{attribute 'qualified_only'}
VAR_GLOBAL
	fJoystickLeftNormalizedY 		: LREAL;
	fJoystickLeftNormalizedX 		: LREAL;
	
	fJoystickRightNormalizedY 		: LREAL;
	fJoystickRightNormalizedX 		: LREAL;
	
	
	//fPositionCylPiston  		: LREAL;
	MCDirectionAxis1 : MC_Direction;
	MCDirectionAxis2 : MC_Direction;
	MCDirectionAxis3 : MC_Direction;
	MCDirectionAxis4 : MC_Direction;
	
		
END_VAR

(* stored: Version 1.1.0.1, ProductVersion 3.1.4024.12
   GVL G_Sensors: Id {d28c946e-63b0-41ab-8fee-be9b6a0df66e} *)
